// TIA Portal V17 export
// export: Created 2023-12-22T15:03:18.8075819Z, ExportSetting WithDefaults, DisplayName Totally Integrated Automation Portal, DisplayVersion V17, DisplayName TIA Portal Openness, DisplayVersion V17, DisplayName TIA Portal Version Control Interface, DisplayVersion V17, DisplayName STEP 7 Professional, DisplayVersion V17, DisplayName STEP 7 Safety, DisplayVersion V17, DisplayName WinCC Advanced, DisplayVersion V17
DATA_BLOCK "Put_Get_DB"   // DB2
VERSION : 0.1
// stored: AutoNumber true, DBAccessibleFromOPCUA true, DBAccessibleFromWebserver true, InstanceOfName Put_Get, InstanceOfType FB
"Put_Get"
   // VAR
   //    GET_SKV_1 { S7_SetPoint := 'True'} : GET;
   //    GET_SKV_2 { S7_SetPoint := 'True'} : GET;
   //    GET_SKV_3 { S7_SetPoint := 'True'} : GET;
   //    GET_SKV_12 { S7_SetPoint := 'True'} : GET;
   //    GET_SKV_13 { S7_SetPoint := 'True'} : GET;
   //    GET_SKV_14 { S7_SetPoint := 'True'} : GET;
   //    GET_SKV_15 { S7_SetPoint := 'True'} : GET;
   //    GET_SKV_20 { S7_SetPoint := 'True'} : GET;
   //    GET_SKV_21 { S7_SetPoint := 'True'} : GET;
   //    GET_SKV_22 { S7_SetPoint := 'True'} : GET;
   //    GET_SKV_23 { S7_SetPoint := 'True'} : GET;
   //    PUT_SKV_1 { S7_SetPoint := 'True'} : PUT;
   //    PUT_SKV_2 { S7_SetPoint := 'True'} : PUT;
   //    PUT_SKV_3 { S7_SetPoint := 'True'} : PUT;
   //    PUT_SKV_12 { S7_SetPoint := 'True'} : PUT;
   //    PUT_SKV_13 { S7_SetPoint := 'True'} : PUT;
   //    PUT_SKV_14 { S7_SetPoint := 'True'} : PUT;
   //    PUT_SKV_15 { S7_SetPoint := 'True'} : PUT;
   //    PUT_SKV_20 { S7_SetPoint := 'True'} : PUT;
   //    PUT_SKV_21 { S7_SetPoint := 'True'} : PUT;
   //    PUT_SKV_22 { S7_SetPoint := 'True'} : PUT;
   //    PUT_SKV_23 { S7_SetPoint := 'True'} : PUT;
   //    GET_SKD2 { S7_SetPoint := 'True'} : GET;
   //    PUT_SKD2 { S7_SetPoint := 'True'} : PUT;
   // END_VAR
BEGIN
END_DATA_BLOCK
